SUBAPPLICATION GreenWhiteBackground2_AX (* Hintergrundfarbe (TRUE -> Grün, FALSE -> Weiß) für 2 Objekte (AX-Adapter) *)
  (* Standard: 61499-2 *)
  (* Version 1.0, 2022-11-10, Franz Höpfinger, Meisterschulen am Ostbahnhof *)
  PACKAGE MyLib::sys;
  IMPORT isobus::UT::Q::const::IDs::ID_NULL;
  IMPORT isobus::UT::Q::const::colours::COLOR_WHITE;
  IMPORT isobus::UT::Q::const::colours::COLOR_GREEN;
  (* Documentation:
  Hintergrundfarbe für ein Auxiliary-Function-Objekt (VT + Aux-Handle)
   Setzt die Hintergrundfarbe (TRUE -> Grün, FALSE -> Weiß) eines Auxiliary-Function-Type-2-Objekts (Object-ID-Bereich 31000–31999) über dieselbe u16ObjIdA an zwei Empfänger gleichzeitig, weil die Zuweisung eines solchen Objekts an zwei Stellen angezeigt wird:
    - VT-Bildschirm (Q_BackgroundColour_1, FB Q_BackgroundColour): die Vorschau der Aux-Zuweisung im Objekt-Pool.
   - Aux-Handle selbst (Q_BackgroundColour_2, FB Q_BackgroundColourAux): die Anzeige am physischen Eingabegerät (z.B. Joystick), das über seine eigene Auxiliary-Connection zum VT-Client separat angesprochen werden muss.
    Beide FBs senden das exakt gleiche ISO-11783-6-Kommando (Part 6 - F.20, "Change Background Colour") mit identischem Interface und identischen gültigen Object-ID-Bereichen - der einzige Unterschied ist die Verbindung, über die es geschickt wird. Für normale VT-Objekte (SoftKeys, Buttons, Output-Felder usw.), die keine eigene Aux-Verbindung haben, genügt dagegen GreenWhiteBackground1_AX mit nur einem Q_BackgroundColour. Für ein normales Objekt UND ein Aux-Objekt gemeinsam (z.B. SoftKey und Joystick lösen dieselbe Funktion aus) GreenWhiteBackground3_AX verwenden.
  *)
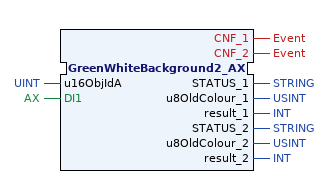
  EVENT_OUTPUT
    CNF_1;
    CNF_2;
  END_EVENT
  VAR_INPUT
    u16ObjIdA : UINT := ID_NULL; (* Object ID AUX *)
  END_VAR
  VAR_OUTPUT
    STATUS_1 : STRING; (* Service Status *)
    u8OldColour_1 : USINT; (* Old value of ID *)
    result_1 : INT; (* retval see description *)
    STATUS_2 : STRING; (* Service Status *)
    u8OldColour_2 : USINT; (* Old value of ID *)
    result_2 : INT; (* retval see description *)
  END_VAR
  SOCKETS
    DI1 : adapter::types::unidirectional::AX; (* Selector *)
  END_SOCKETS
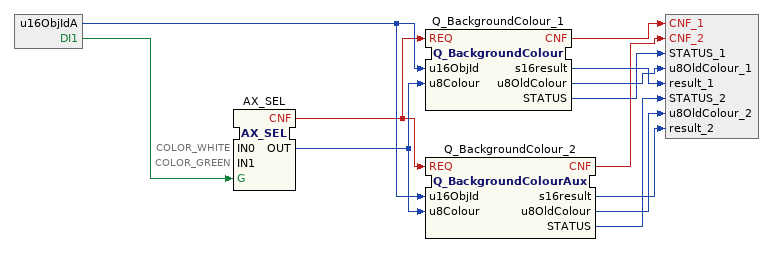
  FBS
    Q_BackgroundColour_1 : isobus::UT::Q::Q_BackgroundColour;
    Q_BackgroundColour_2 : isobus::UT::Q::Q_BackgroundColourAux;
    AX_SEL : adapter::iec61131::selection::AX_SEL(IN0 := COLOR_WHITE, IN1 := COLOR_GREEN);
  END_FBS
  EVENT_CONNECTIONS
    Q_BackgroundColour_1.CNF TO CNF_1;
    Q_BackgroundColour_2.CNF TO CNF_2;
    AX_SEL.CNF TO Q_BackgroundColour_1.REQ;
    AX_SEL.CNF TO Q_BackgroundColour_2.REQ;
  END_CONNECTIONS
  DATA_CONNECTIONS
    u16ObjIdA TO Q_BackgroundColour_1.u16ObjId;
    Q_BackgroundColour_1.s16result TO result_1;
    Q_BackgroundColour_1.u8OldColour TO u8OldColour_1;
    Q_BackgroundColour_1.STATUS TO STATUS_1;
    AX_SEL.OUT TO Q_BackgroundColour_1.u8Colour;
    u16ObjIdA TO Q_BackgroundColour_2.u16ObjId;
    Q_BackgroundColour_2.s16result TO result_2;
    Q_BackgroundColour_2.u8OldColour TO u8OldColour_2;
    Q_BackgroundColour_2.STATUS TO STATUS_2;
    AX_SEL.OUT TO Q_BackgroundColour_2.u8Colour;
  END_CONNECTIONS
  ADAPTER_CONNECTIONS
    DI1 TO AX_SEL.G;
  END_CONNECTIONS
END_SUBAPPLICATION
